FUNCTION alg_a_gripperclose : BOOL
VAR_INPUT
	state: STATE;
END_VAR

alg_a_gripperclose := state.dvar_M_example_controller_a_gripperclose;

END_FUNCTION

(* stored: Version 1.1.0.1, ProductVersion 3.1.4022.18
   POU alg_a_gripperclose: Id {9a06f6e8-4557-489d-b99e-5b3bf56a1417}, SpecialFunc None *)
